  ELSIF iw_cfg_cmd = 1 THEN
    (* --- Write one station to g_stations array --- *)
    IF (iw_cfg_param >= 101) AND (iw_cfg_param <= 125) THEN
      g_stations[iw_cfg_param].tank_id       := iw_cfg_d0;
      g_stations[iw_cfg_param].x_position    := INT_TO_REAL(iw_cfg_d1);
      g_stations[iw_cfg_param].y_position    := INT_TO_REAL(iw_cfg_d2);
      g_stations[iw_cfg_param].z_position    := INT_TO_REAL(iw_cfg_d3);
      g_stations[iw_cfg_param].stn_type      := iw_cfg_d4;
      g_stations[iw_cfg_param].dropping_time := INT_TO_REAL(iw_cfg_d5) / 10.0;
      g_stations[iw_cfg_param].device_delay  := INT_TO_REAL(iw_cfg_d6) / 10.0;
    END_IF;
    qw_cfg_ack := iw_cfg_seq;

  ELSIF iw_cfg_cmd = 2 THEN
    (* --- Finish init: station data uploaded, now init transporters --- *)
    g_station_count := iw_cfg_param;

    (* Transporter 1 config — hardcoded for now *)
    g_cfg[1].x_min_limit := 100.0;
    g_cfg[1].x_max_limit := 20600.0;
    g_cfg[1].x_avoid_mm := 2000.0;
    g_cfg[1].phys2d.x_accel_s := 1.5;
    g_cfg[1].phys2d.x_decel_s := 1.5;
    g_cfg[1].phys2d.x_max_mm_s := 500.0;
    g_cfg[1].phys2d.z_total_mm := 2500.0;
    g_cfg[1].phys2d.z_slow_dry_mm := 300.0;
    g_cfg[1].phys2d.z_slow_wet_mm := 1000.0;
    g_cfg[1].phys2d.z_slow_end_mm := 50.0;
    g_cfg[1].phys2d.z_slow_mm_s := 100.0;
    g_cfg[1].phys2d.z_fast_mm_s := 200.0;
    g_cfg[1].phys2d.drip_delay_s := 5.0;
    g_cfg[1].phys2d.avoid_mm := 2000.0;
    g_cfg[1].task_area[1].min_lift := 101;
    g_cfg[1].task_area[1].max_lift := 111;
    g_cfg[1].task_area[1].min_sink := 101;
    g_cfg[1].task_area[1].max_sink := 114;

    (* Transporter 2 config *)
    g_cfg[2].x_min_limit := 14300.0;
    g_cfg[2].x_max_limit := 29100.0;
    g_cfg[2].x_avoid_mm := 2000.0;
    g_cfg[2].phys2d.x_accel_s := 1.5;
    g_cfg[2].phys2d.x_decel_s := 1.5;
    g_cfg[2].phys2d.x_max_mm_s := 500.0;
    g_cfg[2].phys2d.z_total_mm := 2500.0;
    g_cfg[2].phys2d.z_slow_dry_mm := 300.0;
    g_cfg[2].phys2d.z_slow_wet_mm := 1000.0;
    g_cfg[2].phys2d.z_slow_end_mm := 50.0;
    g_cfg[2].phys2d.z_slow_mm_s := 100.0;
    g_cfg[2].phys2d.z_fast_mm_s := 200.0;
    g_cfg[2].phys2d.drip_delay_s := 5.0;
    g_cfg[2].phys2d.avoid_mm := 2000.0;
    g_cfg[2].task_area[1].min_lift := 112;
    g_cfg[2].task_area[1].max_lift := 121;
    g_cfg[2].task_area[1].min_sink := 111;
    g_cfg[2].task_area[1].max_sink := 121;

    (* Init transporter states *)
    FOR i := 1 TO 3 DO
      IF i <= 2 THEN
        g_state[i].active := TRUE;
      ELSE
        g_state[i].active := FALSE;
      END_IF;
      g_state[i].phase := 0;
      g_state[i].z_stage := 0;
      g_state[i].vel_x := 0.0;
      g_state[i].vel_z := 0.0;
      g_state[i].z_timer_s := 0.0;
      g_state[i].x_min_limit := g_cfg[i].x_min_limit;
      g_state[i].x_max_limit := g_cfg[i].x_max_limit;

      (* Start position: use task_area[1].min_lift as start station *)
      IF g_cfg[i].task_area[1].min_lift > 0 THEN
        stn_num := g_cfg[i].task_area[1].min_lift;
      ELSE
        stn_num := 0;
      END_IF;
      lookup(station_number := stn_num);
      IF lookup.found THEN
        g_state[i].x_mm := lookup.x_mm;
        g_state[i].current_station := stn_num;
      ELSE
        g_state[i].x_mm := 0.0;
        g_state[i].current_station := 0;
      END_IF;
      g_state[i].z_mm := 0.0;
    END_FOR;

    init_done := TRUE;
    qw_cfg_ack := iw_cfg_seq;
  END_IF;
END_IF;

(* ============================================================
   MAIN TRANSPORT CYCLE — only runs when init_done
   ============================================================ *)
IF init_done THEN

(* Calculate transporter working areas (X-limits) every cycle *)
twa_calc();

(* ── Epoch-offset time decode ── *)
(* Server writes iw_epoch_h, iw_time_hi, iw_time_lo via Modbus.
   g_time_s = (iw_time_hi * 65536 + iw_time_lo) / 10.0 *)
g_epoch_h := iw_epoch_h;
g_time_s  := (INT_TO_REAL(iw_time_hi) * 65536.0 + INT_TO_REAL(iw_time_lo)) / 10.0;

(* ── Task Scheduler ── *)
tsk_sched(i_run := init_done, i_time_s := g_time_s);

(* ── Departure Scheduler ── *)
(* Stable signal: TSK is at READY (10000) or RESTART (10110) *)
g_dep_stable := (tsk_sched.o_phase >= 10000);
dep_sched(i_run := init_done, i_time_s := g_time_s, i_tsk_phase := tsk_sched.o_phase);

FOR i := 1 TO 3 DO
  IF g_state[i].active THEN

  IF (g_state[i].phase = 0) AND g_cmd_start[i] THEN
    g_state[i].lift_station_target := g_cmd_lift_station[i];
    g_state[i].sink_station_target := g_cmd_sink_station[i];
    lookup(station_number := g_state[i].lift_station_target);
    g_state[i].target_x := lookup.x_mm;
    g_state[i].phase := 1;
    g_state[i].z_stage := 0;
    g_state[i].z_timer_s := 0.0;
  END_IF;

  IF g_state[i].phase = 1 THEN
    tmp_x := g_state[i].x_mm;
    tmp_vx := g_state[i].vel_x;
    IF i = 1 THEN
      fb_x1(
        delta_t := 0.02,
        x_target := g_state[i].target_x,
        x_min := g_state[i].x_min_limit,
        x_max := g_state[i].x_max_limit,
        v_max := g_cfg[i].phys2d.x_max_mm_s,
        t_acc := g_cfg[i].phys2d.x_accel_s,
        t_dec := g_cfg[i].phys2d.x_decel_s,
        x_pos := tmp_x,
        v_x := tmp_vx
      );
      arrived_x := fb_x1.arrived;
    ELSIF i = 2 THEN
      fb_x2(
        delta_t := 0.02,
        x_target := g_state[i].target_x,
        x_min := g_state[i].x_min_limit,
        x_max := g_state[i].x_max_limit,
        v_max := g_cfg[i].phys2d.x_max_mm_s,
        t_acc := g_cfg[i].phys2d.x_accel_s,
        t_dec := g_cfg[i].phys2d.x_decel_s,
        x_pos := tmp_x,
        v_x := tmp_vx
      );
      arrived_x := fb_x2.arrived;
    ELSIF i = 3 THEN
      fb_x3(
        delta_t := 0.02,
        x_target := g_state[i].target_x,
        x_min := g_state[i].x_min_limit,
        x_max := g_state[i].x_max_limit,
        v_max := g_cfg[i].phys2d.x_max_mm_s,
        t_acc := g_cfg[i].phys2d.x_accel_s,
        t_dec := g_cfg[i].phys2d.x_decel_s,
        x_pos := tmp_x,
        v_x := tmp_vx
      );
      arrived_x := fb_x3.arrived;
    END_IF;
    g_state[i].x_mm := tmp_x;
    g_state[i].vel_x := tmp_vx;

    IF arrived_x THEN
      g_state[i].current_station := g_state[i].lift_station_target;
      lookup(station_number := g_state[i].lift_station_target);
      device_delay := lookup.device_delay_s;
      drop_time := lookup.dropping_time_s;
      g_state[i].z_timer_s := device_delay + drop_time;
      g_state[i].z_stage := 1;
      g_state[i].phase := 2;
    END_IF;
  END_IF;

  IF g_state[i].phase = 2 THEN
    lookup(station_number := g_state[i].lift_station_target);
    station_type := lookup.stype;
    tmp_z := g_state[i].z_mm;
    tmp_zs := g_state[i].z_stage;
    tmp_zt := g_state[i].z_timer_s;
    IF i = 1 THEN
      fb_z1(
        delta_t := 0.02,
        station_type := station_type,
        z_total_mm := g_cfg[i].phys2d.z_total_mm,
        z_slow_dry_mm := g_cfg[i].phys2d.z_slow_dry_mm,
        z_slow_wet_mm := g_cfg[i].phys2d.z_slow_wet_mm,
        z_slow_end_mm := g_cfg[i].phys2d.z_slow_end_mm,
        z_slow_mm_s := g_cfg[i].phys2d.z_slow_mm_s,
        z_fast_mm_s := g_cfg[i].phys2d.z_fast_mm_s,
        drip_delay_s := g_cfg[i].phys2d.drip_delay_s,
        z_mm := tmp_z,
        z_stage := tmp_zs,
        z_timer_s := tmp_zt
      );
      arrived_z := fb_z1.done;
    ELSIF i = 2 THEN
      fb_z2(
        delta_t := 0.02,
        station_type := station_type,
        z_total_mm := g_cfg[i].phys2d.z_total_mm,
        z_slow_dry_mm := g_cfg[i].phys2d.z_slow_dry_mm,
        z_slow_wet_mm := g_cfg[i].phys2d.z_slow_wet_mm,
        z_slow_end_mm := g_cfg[i].phys2d.z_slow_end_mm,
        z_slow_mm_s := g_cfg[i].phys2d.z_slow_mm_s,
        z_fast_mm_s := g_cfg[i].phys2d.z_fast_mm_s,
        drip_delay_s := g_cfg[i].phys2d.drip_delay_s,
        z_mm := tmp_z,
        z_stage := tmp_zs,
        z_timer_s := tmp_zt
      );
      arrived_z := fb_z2.done;
    ELSIF i = 3 THEN
      fb_z3(
        delta_t := 0.02,
        station_type := station_type,
        z_total_mm := g_cfg[i].phys2d.z_total_mm,
        z_slow_dry_mm := g_cfg[i].phys2d.z_slow_dry_mm,
        z_slow_wet_mm := g_cfg[i].phys2d.z_slow_wet_mm,
        z_slow_end_mm := g_cfg[i].phys2d.z_slow_end_mm,
        z_slow_mm_s := g_cfg[i].phys2d.z_slow_mm_s,
        z_fast_mm_s := g_cfg[i].phys2d.z_fast_mm_s,
        drip_delay_s := g_cfg[i].phys2d.drip_delay_s,
        z_mm := tmp_z,
        z_stage := tmp_zs,
        z_timer_s := tmp_zt
      );
      arrived_z := fb_z3.done;
    END_IF;
    g_state[i].z_mm := tmp_z;
    g_state[i].z_stage := tmp_zs;
    g_state[i].z_timer_s := tmp_zt;
    IF arrived_z THEN
      lookup(station_number := g_state[i].sink_station_target);
      g_state[i].target_x := lookup.x_mm;
      g_state[i].phase := 3;
    END_IF;
  END_IF;

  IF g_state[i].phase = 3 THEN
    tmp_x := g_state[i].x_mm;
    tmp_vx := g_state[i].vel_x;
    IF i = 1 THEN
      fb_x1(
        delta_t := 0.02,
        x_target := g_state[i].target_x,
        x_min := g_state[i].x_min_limit,
        x_max := g_state[i].x_max_limit,
        v_max := g_cfg[i].phys2d.x_max_mm_s,
        t_acc := g_cfg[i].phys2d.x_accel_s,
        t_dec := g_cfg[i].phys2d.x_decel_s,
        x_pos := tmp_x,
        v_x := tmp_vx
      );
      arrived_x := fb_x1.arrived;
    ELSIF i = 2 THEN
      fb_x2(
        delta_t := 0.02,
        x_target := g_state[i].target_x,
        x_min := g_state[i].x_min_limit,
        x_max := g_state[i].x_max_limit,
        v_max := g_cfg[i].phys2d.x_max_mm_s,
        t_acc := g_cfg[i].phys2d.x_accel_s,
        t_dec := g_cfg[i].phys2d.x_decel_s,
        x_pos := tmp_x,
        v_x := tmp_vx
      );
      arrived_x := fb_x2.arrived;
    ELSIF i = 3 THEN
      fb_x3(
        delta_t := 0.02,
        x_target := g_state[i].target_x,
        x_min := g_state[i].x_min_limit,
        x_max := g_state[i].x_max_limit,
        v_max := g_cfg[i].phys2d.x_max_mm_s,
        t_acc := g_cfg[i].phys2d.x_accel_s,
        t_dec := g_cfg[i].phys2d.x_decel_s,
        x_pos := tmp_x,
        v_x := tmp_vx
      );
      arrived_x := fb_x3.arrived;
    END_IF;
    g_state[i].x_mm := tmp_x;
    g_state[i].vel_x := tmp_vx;

    IF arrived_x THEN
      g_state[i].current_station := g_state[i].sink_station_target;
      lookup(station_number := g_state[i].sink_station_target);
      device_delay := lookup.device_delay_s;
      g_state[i].z_timer_s := device_delay + g_cfg[i].phys2d.drip_delay_s;
      g_state[i].z_stage := 6;
      g_state[i].phase := 4;
    END_IF;
  END_IF;

  IF g_state[i].phase = 4 THEN
    lookup(station_number := g_state[i].sink_station_target);
    station_type := lookup.stype;
    tmp_z := g_state[i].z_mm;
    tmp_zs := g_state[i].z_stage;
    tmp_zt := g_state[i].z_timer_s;
    IF i = 1 THEN
      fb_z1(
        delta_t := 0.02,
        station_type := station_type,
        z_total_mm := g_cfg[i].phys2d.z_total_mm,
        z_slow_dry_mm := g_cfg[i].phys2d.z_slow_dry_mm,
        z_slow_wet_mm := g_cfg[i].phys2d.z_slow_wet_mm,
        z_slow_end_mm := g_cfg[i].phys2d.z_slow_end_mm,
        z_slow_mm_s := g_cfg[i].phys2d.z_slow_mm_s,
        z_fast_mm_s := g_cfg[i].phys2d.z_fast_mm_s,
        drip_delay_s := g_cfg[i].phys2d.drip_delay_s,
        z_mm := tmp_z,
        z_stage := tmp_zs,
        z_timer_s := tmp_zt
      );
      arrived_z := fb_z1.done;
    ELSIF i = 2 THEN
      fb_z2(
        delta_t := 0.02,
        station_type := station_type,
        z_total_mm := g_cfg[i].phys2d.z_total_mm,
        z_slow_dry_mm := g_cfg[i].phys2d.z_slow_dry_mm,
        z_slow_wet_mm := g_cfg[i].phys2d.z_slow_wet_mm,
        z_slow_end_mm := g_cfg[i].phys2d.z_slow_end_mm,
        z_slow_mm_s := g_cfg[i].phys2d.z_slow_mm_s,
        z_fast_mm_s := g_cfg[i].phys2d.z_fast_mm_s,
        drip_delay_s := g_cfg[i].phys2d.drip_delay_s,
        z_mm := tmp_z,
        z_stage := tmp_zs,
        z_timer_s := tmp_zt
      );
      arrived_z := fb_z2.done;
    ELSIF i = 3 THEN
      fb_z3(
        delta_t := 0.02,
        station_type := station_type,
        z_total_mm := g_cfg[i].phys2d.z_total_mm,
        z_slow_dry_mm := g_cfg[i].phys2d.z_slow_dry_mm,
        z_slow_wet_mm := g_cfg[i].phys2d.z_slow_wet_mm,
        z_slow_end_mm := g_cfg[i].phys2d.z_slow_end_mm,
        z_slow_mm_s := g_cfg[i].phys2d.z_slow_mm_s,
        z_fast_mm_s := g_cfg[i].phys2d.z_fast_mm_s,
        drip_delay_s := g_cfg[i].phys2d.drip_delay_s,
        z_mm := tmp_z,
        z_stage := tmp_zs,
        z_timer_s := tmp_zt
      );
      arrived_z := fb_z3.done;
    END_IF;
    g_state[i].z_mm := tmp_z;
    g_state[i].z_stage := tmp_zs;
    g_state[i].z_timer_s := tmp_zt;
    IF arrived_z THEN
      g_state[i].phase := 0;
    END_IF;
  END_IF;

  min_dist := 1.0e9;
  nearest_num := g_state[i].current_station;
  FOR idx := 101 TO 125 DO
    IF g_stations[idx].tank_id <> 0 THEN
      dx := g_stations[idx].x_position - g_state[i].x_mm;
      IF ABS(dx) < min_dist THEN
        min_dist := ABS(dx);
        nearest_num := idx;
      END_IF;
    END_IF;
  END_FOR;
  g_state[i].current_station := nearest_num;

  END_IF;  (* active *)
END_FOR;

END_IF;  (* init_done *)

(* ============================================================
   UNIT WRITE HANDLER — gateway writes one unit at a time
   ============================================================ *)
IF iw_unit_seq <> last_unit_seq THEN
  last_unit_seq := iw_unit_seq;
  IF (iw_unit_id >= 1) AND (iw_unit_id <= 10) THEN
    g_units[iw_unit_id].location := iw_unit_loc;
    g_units[iw_unit_id].status   := iw_unit_status;
    g_units[iw_unit_id].state    := iw_unit_state;
    g_units[iw_unit_id].target   := iw_unit_target;
  END_IF;
  qw_unit_ack := iw_unit_seq;
END_IF;

(* ============================================================
   BATCH WRITE HANDLER — gateway writes batch data + program_id
   Also clears all stages of the treatment program for this unit.
   ============================================================ *)
IF iw_batch_seq <> last_batch_seq THEN
  last_batch_seq := iw_batch_seq;
  IF (iw_batch_unit >= 1) AND (iw_batch_unit <= 10) THEN
    g_batches[iw_batch_unit].batch_code := iw_batch_code;
    g_batches[iw_batch_unit].state      := iw_batch_state;
    g_batches[iw_batch_unit].prog_id    := iw_batch_prog_id;
    g_batches[iw_batch_unit].cur_stage      := 0;
    g_programs[iw_batch_unit].program_id := iw_batch_prog_id;
    (* Clear all stages *)
    FOR j := 1 TO 30 DO
      FOR k := 1 TO 5 DO
        g_programs[iw_batch_unit].stages[j].stations[k] := 0;
      END_FOR;
      g_programs[iw_batch_unit].stages[j].min_time := 0;
      g_programs[iw_batch_unit].stages[j].max_time := 0;
      g_programs[iw_batch_unit].stages[j].cal_time := 0;
    END_FOR;
  END_IF;
  qw_batch_ack := iw_batch_seq;
END_IF;

(* ============================================================
   PROGRAM STAGE WRITE HANDLER — gateway writes one stage at a time
   ============================================================ *)
IF iw_prog_seq <> last_prog_seq THEN
  last_prog_seq := iw_prog_seq;
  IF (iw_prog_unit >= 1) AND (iw_prog_unit <= 10) AND
     (iw_prog_stage >= 1) AND (iw_prog_stage <= 30) THEN
    g_programs[iw_prog_unit].stages[iw_prog_stage].stations[1] := iw_prog_s1;
    g_programs[iw_prog_unit].stages[iw_prog_stage].stations[2] := iw_prog_s2;
    g_programs[iw_prog_unit].stages[iw_prog_stage].stations[3] := iw_prog_s3;
    g_programs[iw_prog_unit].stages[iw_prog_stage].stations[4] := iw_prog_s4;
    g_programs[iw_prog_unit].stages[iw_prog_stage].stations[5] := iw_prog_s5;
    g_programs[iw_prog_unit].stages[iw_prog_stage].min_time := iw_prog_min_time;
    g_programs[iw_prog_unit].stages[iw_prog_stage].max_time := iw_prog_max_time;
    g_programs[iw_prog_unit].stages[iw_prog_stage].cal_time := iw_prog_cal_time;
  END_IF;
  qw_prog_ack := iw_prog_seq;
END_IF;

(* === MODBUS INPUT: Read commands from input registers === *)
g_cmd_start[1] := iw_cmd_start_1 <> 0;
g_cmd_lift_station[1] := iw_cmd_lift_1;
g_cmd_sink_station[1] := iw_cmd_sink_1;
g_cmd_start[2] := iw_cmd_start_2 <> 0;
g_cmd_lift_station[2] := iw_cmd_lift_2;
g_cmd_sink_station[2] := iw_cmd_sink_2;

(* === MODBUS OUTPUT: Write transporter 1 state === *)
qw_t1_x_mm := REAL_TO_INT(g_state[1].x_mm);
qw_t1_z_mm := REAL_TO_INT(g_state[1].z_mm);
qw_t1_vel_x10 := REAL_TO_INT(g_state[1].vel_x * 10.0);
qw_t1_phase := g_state[1].phase;
qw_t1_z_stage := g_state[1].z_stage;
qw_t1_cur_st := g_state[1].current_station;
qw_t1_lift_tgt := g_state[1].lift_station_target;
qw_t1_sink_tgt := g_state[1].sink_station_target;
IF g_state[1].active THEN qw_t1_active := 1; ELSE qw_t1_active := 0; END_IF;

(* === MODBUS OUTPUT: Write transporter 2 state === *)
qw_t2_x_mm := REAL_TO_INT(g_state[2].x_mm);
qw_t2_z_mm := REAL_TO_INT(g_state[2].z_mm);
qw_t2_vel_x10 := REAL_TO_INT(g_state[2].vel_x * 10.0);
qw_t2_phase := g_state[2].phase;
qw_t2_z_stage := g_state[2].z_stage;
qw_t2_cur_st := g_state[2].current_station;
qw_t2_lift_tgt := g_state[2].lift_station_target;
qw_t2_sink_tgt := g_state[2].sink_station_target;
IF g_state[2].active THEN qw_t2_active := 1; ELSE qw_t2_active := 0; END_IF;

(* === MODBUS OUTPUT: Status registers === *)
qw_station_cnt := g_station_count;
IF init_done THEN qw_init_done := 1; ELSE qw_init_done := 0; END_IF;
cycle_count := cycle_count + 1;
IF cycle_count > 30000 THEN cycle_count := 0; END_IF;
qw_cycle_cnt := cycle_count;

(* Write unit data to Modbus output QW22..QW61 *)
qw_u1_loc    := g_units[1].location;
qw_u1_status := g_units[1].status;
qw_u1_state  := g_units[1].state;
qw_u1_target := g_units[1].target;
qw_u2_loc    := g_units[2].location;
qw_u2_status := g_units[2].status;
qw_u2_state  := g_units[2].state;
qw_u2_target := g_units[2].target;
qw_u3_loc    := g_units[3].location;
qw_u3_status := g_units[3].status;
qw_u3_state  := g_units[3].state;
qw_u3_target := g_units[3].target;
qw_u4_loc    := g_units[4].location;
qw_u4_status := g_units[4].status;
qw_u4_state  := g_units[4].state;
qw_u4_target := g_units[4].target;
qw_u5_loc    := g_units[5].location;
qw_u5_status := g_units[5].status;
qw_u5_state  := g_units[5].state;
qw_u5_target := g_units[5].target;
qw_u6_loc    := g_units[6].location;
qw_u6_status := g_units[6].status;
qw_u6_state  := g_units[6].state;
qw_u6_target := g_units[6].target;
qw_u7_loc    := g_units[7].location;
qw_u7_status := g_units[7].status;
qw_u7_state  := g_units[7].state;
qw_u7_target := g_units[7].target;
qw_u8_loc    := g_units[8].location;
qw_u8_status := g_units[8].status;
qw_u8_state  := g_units[8].state;
qw_u8_target := g_units[8].target;
qw_u9_loc    := g_units[9].location;
qw_u9_status := g_units[9].status;
qw_u9_state  := g_units[9].state;
qw_u9_target := g_units[9].target;
qw_u10_loc    := g_units[10].location;
qw_u10_status := g_units[10].status;
qw_u10_state  := g_units[10].state;
qw_u10_target := g_units[10].target;

(* Write batch data to Modbus output QW65..QW104 *)
qw_b1_code  := g_batches[1].batch_code;  qw_b1_state  := g_batches[1].state;  qw_b1_prog  := g_batches[1].prog_id;  qw_b1_stage  := g_batches[1].cur_stage;
qw_b2_code  := g_batches[2].batch_code;  qw_b2_state  := g_batches[2].state;  qw_b2_prog  := g_batches[2].prog_id;  qw_b2_stage  := g_batches[2].cur_stage;
qw_b3_code  := g_batches[3].batch_code;  qw_b3_state  := g_batches[3].state;  qw_b3_prog  := g_batches[3].prog_id;  qw_b3_stage  := g_batches[3].cur_stage;
qw_b4_code  := g_batches[4].batch_code;  qw_b4_state  := g_batches[4].state;  qw_b4_prog  := g_batches[4].prog_id;  qw_b4_stage  := g_batches[4].cur_stage;
qw_b5_code  := g_batches[5].batch_code;  qw_b5_state  := g_batches[5].state;  qw_b5_prog  := g_batches[5].prog_id;  qw_b5_stage  := g_batches[5].cur_stage;
qw_b6_code  := g_batches[6].batch_code;  qw_b6_state  := g_batches[6].state;  qw_b6_prog  := g_batches[6].prog_id;  qw_b6_stage  := g_batches[6].cur_stage;
qw_b7_code  := g_batches[7].batch_code;  qw_b7_state  := g_batches[7].state;  qw_b7_prog  := g_batches[7].prog_id;  qw_b7_stage  := g_batches[7].cur_stage;
qw_b8_code  := g_batches[8].batch_code;  qw_b8_state  := g_batches[8].state;  qw_b8_prog  := g_batches[8].prog_id;  qw_b8_stage  := g_batches[8].cur_stage;
qw_b9_code  := g_batches[9].batch_code;  qw_b9_state  := g_batches[9].state;  qw_b9_prog  := g_batches[9].prog_id;  qw_b9_stage  := g_batches[9].cur_stage;
qw_b10_code := g_batches[10].batch_code; qw_b10_state := g_batches[10].state; qw_b10_prog := g_batches[10].prog_id; qw_b10_stage := g_batches[10].cur_stage;
          
END_PROGRAM

CONFIGURATION Config0
  VAR_GLOBAL
    MAX_STATIONS : INT := 25;
    MAX_TRANSPORTERS : INT := 3;
    MAX_UNITS : INT := 10;
    USED : INT := 1;
    NOT_USED : INT := 0;
    EMPTY : INT := 0;
    FULL : INT := 1;
    TO_NONE : INT := 0;
    TO_LOADING : INT := 1;
    TO_BUFFER : INT := 2;
    TO_PROCESS : INT := 3;
    TO_UNLOAD : INT := 4;
    TO_AVOID : INT := 5;
    STN_DRY : INT := 0;
    STN_WET : INT := 1;
    NOT_PROCESSED : INT := 0;
    IN_PROCESS : INT := 1;
    PROCESSED : INT := 2;
    MAX_PARALLELS : INT := 5;
    MAX_STAGES : INT := 30;
    MAX_LINES : INT := 4;
    AVOID_NONE : INT := 0;
    AVOID_PASS : INT := 1;
    AVOID_BLOCK : INT := 2;
    MIN_WORK_AREA : REAL := 1000.0;
    DEP_MAX_IDLE_SLOTS : INT := 20;
    DEP_MAX_DELAY_ACTS : INT := 10;
    DEP_MAX_WAITING : INT := 10;
    g_station_count : INT := 0;
    g_stations : ARRAY[101..125] OF STATION_T;
    g_cfg : ARRAY[1..3] OF TRANSPORTER_CFG_T;
    g_state : ARRAY[1..3] OF TRANSPORTER_STATE_T;
    g_cmd_start : ARRAY[1..3] OF BOOL;
    g_cmd_lift_station : ARRAY[1..3] OF INT;
    g_cmd_sink_station : ARRAY[1..3] OF INT;
    g_units : ARRAY[1..10] OF UNIT_T;
    g_batches : ARRAY[1..10] OF BATCH_T;
    g_programs : ARRAY[1..10] OF TREATMENT_PROGRAM_T;
    g_avoid_status : ARRAY[101..125] OF INT;
    g_move : ARRAY[1..3] OF MOVE_TIMES_T;
    g_schedule : ARRAY[1..10] OF TSK_SCHEDULE_T;
    g_tasks : ARRAY[1..3] OF TSK_QUEUE_T;
    g_dep_sandbox : DEP_SANDBOX_T;
    g_dep_idle_slots : ARRAY[1..3] OF DEP_IDLE_SLOT_SET_T;
    g_dep_waiting : ARRAY[1..10] OF INT;
    g_dep_waiting_count : INT;
    g_dep_overlap : DEP_OVERLAP_T;
    g_dep_pending : DEP_PENDING_WRITE_T;
    g_dep_activated : BOOL;
    g_dep_stable : BOOL;
    g_epoch_h : INT;
    g_time_s : REAL;
    qw_t1_x_mm AT %QW0 : INT;
    qw_t1_z_mm AT %QW1 : INT;
    qw_t1_vel_x10 AT %QW2 : INT;
    qw_t1_phase AT %QW3 : INT;
    qw_t1_z_stage AT %QW4 : INT;
    qw_t1_cur_st AT %QW5 : INT;
    qw_t1_lift_tgt AT %QW6 : INT;
    qw_t1_sink_tgt AT %QW7 : INT;
    qw_t1_active AT %QW8 : INT;
    qw_t2_x_mm AT %QW9 : INT;
    qw_t2_z_mm AT %QW10 : INT;
    qw_t2_vel_x10 AT %QW11 : INT;
    qw_t2_phase AT %QW12 : INT;
    qw_t2_z_stage AT %QW13 : INT;
    qw_t2_cur_st AT %QW14 : INT;
    qw_t2_lift_tgt AT %QW15 : INT;
    qw_t2_sink_tgt AT %QW16 : INT;
    qw_t2_active AT %QW17 : INT;
    qw_station_cnt AT %QW18 : INT;
    qw_init_done AT %QW19 : INT;
    qw_cycle_cnt AT %QW20 : INT;
    qw_b1_code AT %QW65 : INT;
    qw_b1_state AT %QW66 : INT;
    qw_b1_prog AT %QW67 : INT;
    qw_b1_stage AT %QW68 : INT;
    qw_b2_code AT %QW69 : INT;
    qw_b2_state AT %QW70 : INT;
    qw_b2_prog AT %QW71 : INT;
    qw_b2_stage AT %QW72 : INT;
    qw_b3_code AT %QW73 : INT;
    qw_b3_state AT %QW74 : INT;
    qw_b3_prog AT %QW75 : INT;
    qw_b3_stage AT %QW76 : INT;
    qw_b4_code AT %QW77 : INT;
    qw_b4_state AT %QW78 : INT;
    qw_b4_prog AT %QW79 : INT;
    qw_b4_stage AT %QW80 : INT;
    qw_b5_code AT %QW81 : INT;
    qw_b5_state AT %QW82 : INT;
    qw_b5_prog AT %QW83 : INT;
    qw_b5_stage AT %QW84 : INT;
    qw_b6_code AT %QW85 : INT;
    qw_b6_state AT %QW86 : INT;
    qw_b6_prog AT %QW87 : INT;
    qw_b6_stage AT %QW88 : INT;
    qw_b7_code AT %QW89 : INT;
    qw_b7_state AT %QW90 : INT;
    qw_b7_prog AT %QW91 : INT;
    qw_b7_stage AT %QW92 : INT;
    qw_b8_code AT %QW93 : INT;
    qw_b8_state AT %QW94 : INT;
    qw_b8_prog AT %QW95 : INT;
    qw_b8_stage AT %QW96 : INT;
    qw_b9_code AT %QW97 : INT;
    qw_b9_state AT %QW98 : INT;
    qw_b9_prog AT %QW99 : INT;
    qw_b9_stage AT %QW100 : INT;
    qw_b10_code AT %QW101 : INT;
    qw_b10_state AT %QW102 : INT;
    qw_b10_prog AT %QW103 : INT;
    qw_b10_stage AT %QW104 : INT;
    iw_cmd_start_1 AT %QW200 : INT;
    iw_cmd_lift_1 AT %QW201 : INT;
    iw_cmd_sink_1 AT %QW202 : INT;
    iw_cmd_start_2 AT %QW203 : INT;
    iw_cmd_lift_2 AT %QW204 : INT;
    iw_cmd_sink_2 AT %QW205 : INT;
    iw_cfg_seq AT %QW110 : INT;
    iw_cfg_cmd AT %QW111 : INT;
    iw_cfg_param AT %QW112 : INT;
    iw_cfg_d0 AT %QW113 : INT;
    iw_cfg_d1 AT %QW114 : INT;
    iw_cfg_d2 AT %QW115 : INT;
    iw_cfg_d3 AT %QW116 : INT;
    iw_cfg_d4 AT %QW117 : INT;
    iw_cfg_d5 AT %QW118 : INT;
    iw_cfg_d6 AT %QW119 : INT;
    qw_cfg_ack AT %QW21 : INT;
    qw_u1_loc AT %QW22 : INT;
    qw_u1_status AT %QW23 : INT;
    qw_u1_state AT %QW24 : INT;
    qw_u1_target AT %QW25 : INT;
    qw_u2_loc AT %QW26 : INT;
    qw_u2_status AT %QW27 : INT;
    qw_u2_state AT %QW28 : INT;
    qw_u2_target AT %QW29 : INT;
    qw_u3_loc AT %QW30 : INT;
    qw_u3_status AT %QW31 : INT;
    qw_u3_state AT %QW32 : INT;
    qw_u3_target AT %QW33 : INT;
    qw_u4_loc AT %QW34 : INT;
    qw_u4_status AT %QW35 : INT;
    qw_u4_state AT %QW36 : INT;
    qw_u4_target AT %QW37 : INT;
    qw_u5_loc AT %QW38 : INT;
    qw_u5_status AT %QW39 : INT;
    qw_u5_state AT %QW40 : INT;
    qw_u5_target AT %QW41 : INT;
    qw_u6_loc AT %QW42 : INT;
    qw_u6_status AT %QW43 : INT;
    qw_u6_state AT %QW44 : INT;
    qw_u6_target AT %QW45 : INT;
    qw_u7_loc AT %QW46 : INT;
    qw_u7_status AT %QW47 : INT;
    qw_u7_state AT %QW48 : INT;
    qw_u7_target AT %QW49 : INT;
    qw_u8_loc AT %QW50 : INT;
    qw_u8_status AT %QW51 : INT;
    qw_u8_state AT %QW52 : INT;
    qw_u8_target AT %QW53 : INT;
    qw_u9_loc AT %QW54 : INT;
    qw_u9_status AT %QW55 : INT;
    qw_u9_state AT %QW56 : INT;
    qw_u9_target AT %QW57 : INT;
    qw_u10_loc AT %QW58 : INT;
    qw_u10_status AT %QW59 : INT;
    qw_u10_state AT %QW60 : INT;
    qw_u10_target AT %QW61 : INT;
    qw_unit_ack AT %QW62 : INT;
    iw_unit_seq AT %QW120 : INT;
    iw_unit_id AT %QW121 : INT;
    iw_unit_loc AT %QW122 : INT;
    iw_unit_status AT %QW123 : INT;
    iw_unit_state AT %QW124 : INT;
    iw_unit_target AT %QW125 : INT;
    iw_batch_seq AT %QW130 : INT;
    iw_batch_unit AT %QW131 : INT;
    iw_batch_code AT %QW132 : INT;
    iw_batch_state AT %QW133 : INT;
    iw_batch_prog_id AT %QW134 : INT;
    qw_batch_ack AT %QW63 : INT;
    iw_prog_seq AT %QW140 : INT;
    iw_prog_unit AT %QW141 : INT;
    iw_prog_stage AT %QW142 : INT;
    iw_prog_s1 AT %QW143 : INT;
    iw_prog_s2 AT %QW144 : INT;
    iw_prog_s3 AT %QW145 : INT;
    iw_prog_s4 AT %QW146 : INT;
    iw_prog_s5 AT %QW147 : INT;
    iw_prog_min_time AT %QW148 : INT;
    iw_prog_max_time AT %QW149 : INT;
    iw_prog_cal_time AT %QW150 : INT;
    qw_prog_ack AT %QW64 : INT;
    iw_epoch_h AT %QW160 : INT;
    iw_time_hi AT %QW161 : INT;
    iw_time_lo AT %QW162 : INT;
  END_VAR
  RESOURCE Res0 ON PLC
    TASK task0(INTERVAL := T#20ms, PRIORITY := 0);
    PROGRAM instance0 WITH task0 : PLC_PRG;
  END_RESOURCE
END_CONFIGURATION
